// TIA Portal V19 export
ORGANIZATION_BLOCK "Startup"   // OB200, LAD, Startup
TITLE = "Complete Restart"
// stored: AutoNumber false, IsIECCheckEnabled true, SetENOAutomatically true
   VAR_INPUT
      LostRetentive : Bool;   // True if retentive data are lost
      LostRTC : Bool;   // True if date and time are lost
   END_VAR
   VAR_TEMP
      tempError : Bool;
      tempStatus : Word;
      tempDiagnostics : "LAF_typeDiagnosticsSimple";
   END_VAR
BEGIN

REGION Network 1: Set first cycle bit / Erster Zyklus bit setzen
   // Set the first cycle signal / Setze das "erster Zyklus" Signal und die Signale immer EIN sowie immer AUS
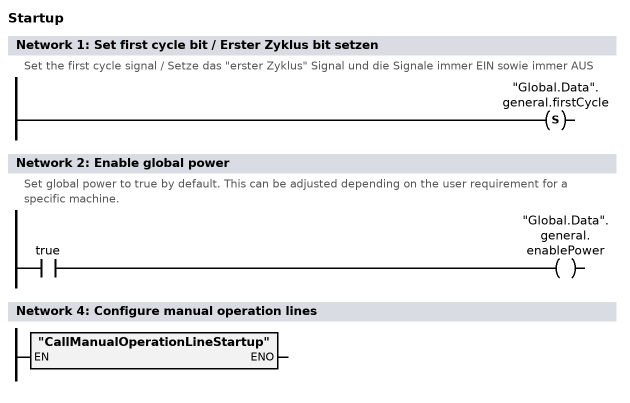
   RUNG wire#powerrail
      S_Coil( "Global.Data".general.firstCycle )
   END_RUNG
   // the same network as SCL:
   "Global.Data".general.firstCycle := TRUE;
END_REGION

REGION Network 2: Enable global power
   // Set global power to true by default. This can be adjusted depending on the user requirement for a specific machine.
   RUNG wire#powerrail
      Contact( true )
      Coil( "Global.Data".general.enablePower )
   END_RUNG
   // the same network as SCL:
   "Global.Data".general.enablePower := true;
END_REGION

REGION Network 3: Set drive objects for drive diagnostic
END_REGION

REGION Network 4: Configure manual operation lines
   RUNG wire#powerrail
      "CallManualOperationLineStartup"()
   END_RUNG
   // the same network as SCL:
   "CallManualOperationLineStartup"();
END_REGION
END_ORGANIZATION_BLOCK
